(* CODESYS project addition_4.xml

Project tree, tasks and I/O mapping:
  function block addition_4 [ST]
*)

// addition_4
FUNCTION_BLOCK addition_4
VAR_INPUT
	yo:BOOL;
END_VAR
VAR_OUTPUT
	yoyo:INT;
END_VAR
VAR
	yoyoyo:STRING;
END_VAR

yo		:=		TRUE;

yoyo	:=		50;

yoyoyo	:=		'HELELELE';

END_FUNCTION_BLOCK
